Staubli VAL3: chkPosStatus.pgx

public program chkPosStatus(bool& x_bIsSame, num x_nAxisNum, num x_nAxisPos)
begin
  //检查外部轴是否在指定位置上
  x_bIsSame=abs(aioGet(aiPosFbk[x_nAxisNum])-x_nAxisPos*nGearratio[x_nAxisNum]*nResolution[x_nAxisNum]/nScaleFact[x_nAxisNum])<=5
end
